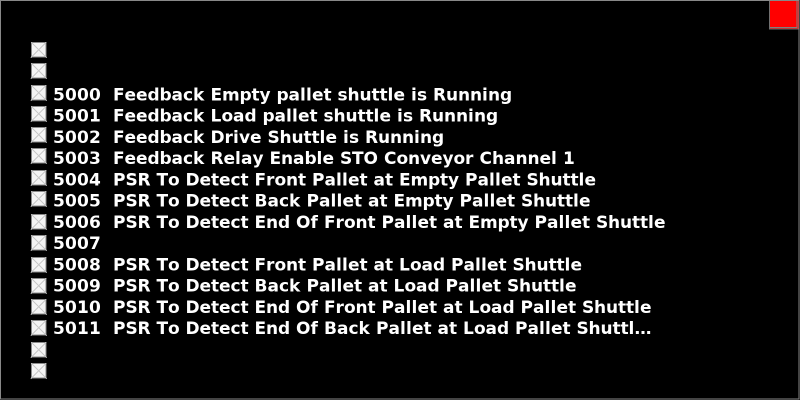
VISUALIZATION P3_DI1  // 800x400, background image 
    ImageSwitcher (31,42 15x15), variable: InputOutput_GVL.Digital_Input[113], behaviour: TOGGLE
    Label (50,16 706x391), "5000 Feedback Empty pallet shuttle is Running 5001 Feedback Load pallet shuttle is Running 5002 Feedback Drive Shuttle is Running 5003 Feedback Relay Enable STO Conveyor Channel 1 5004 PSR To Detect Front Pallet at Empty Pallet Shuttle 5005 PSR To Detect Back Pallet at Empty Pallet Shuttle 5006 PSR To Detect End Of Front Pallet at Empty Pallet Shuttle 5007 5008 PSR To Detect Front Pallet at Load Pallet Shuttle 5009 PSR To Detect Back Pallet at Load Pallet Shuttle 5010 PSR To Detect End Of Front Pallet at Load Pallet Shuttle 5011 PSR To Detect End Of Back Pallet at Load Pallet Shuttle 5012 Limit Switch To Detect Left Limit Area 5013 Limit Switch To Detect Right Limit Area 5014 PRX to Detect Left Limit Area 5015 PRX to Detect Right Limit Area"
    ImageSwitcher (31,63 15x15), variable: InputOutput_GVL.Digital_Input[114], behaviour: TOGGLE
    ImageSwitcher (31,85 15x15), variable: InputOutput_GVL.Digital_Input[115], behaviour: TOGGLE
    ImageSwitcher (31,106 15x15), variable: InputOutput_GVL.Digital_Input[116], behaviour: TOGGLE
    ImageSwitcher (31,127 15x15), variable: InputOutput_GVL.Digital_Input[117], behaviour: TOGGLE
    ImageSwitcher (31,148 15x15), variable: InputOutput_GVL.Digital_Input[118], behaviour: TOGGLE
    ImageSwitcher (31,170 15x15), variable: InputOutput_GVL.Digital_Input[119], behaviour: TOGGLE
    ImageSwitcher (31,191 15x15), variable: InputOutput_GVL.Digital_Input[120], behaviour: TOGGLE
    ImageSwitcher (31,214 15x15), variable: InputOutput_GVL.Digital_Input[121], behaviour: TOGGLE
    ImageSwitcher (31,235 15x15), variable: InputOutput_GVL.Digital_Input[122], behaviour: TOGGLE
    ImageSwitcher (31,257 15x15), variable: InputOutput_GVL.Digital_Input[123], behaviour: TOGGLE
    ImageSwitcher (31,278 15x15), variable: InputOutput_GVL.Digital_Input[124], behaviour: TOGGLE
    ImageSwitcher (31,299 15x15), variable: InputOutput_GVL.Digital_Input[125], behaviour: TOGGLE
    ImageSwitcher (31,320 15x15), variable: InputOutput_GVL.Digital_Input[126], behaviour: TOGGLE
    ImageSwitcher (31,342 15x15), variable: InputOutput_GVL.Digital_Input[127], behaviour: TOGGLE
    ImageSwitcher (31,363 15x15), variable: InputOutput_GVL.Digital_Input[128], behaviour: TOGGLE
    Button (769,-1 30x30), image: VisuSymbols.Symbols.Wrong
        OnMouseClick: CloseDialog Dialog=P3_DI1, Result=OK, NumpadKeypadSet=True
END_VISUALIZATION

(* stored: Version 1.1.0.1, ProductVersion 3.1.4024.12
   Visu P3_DI1: Id {5423823e-5f67-4f8b-af74-d75a729e32c2} *)
